ABB RobotStudio station: Lab1.rsstn

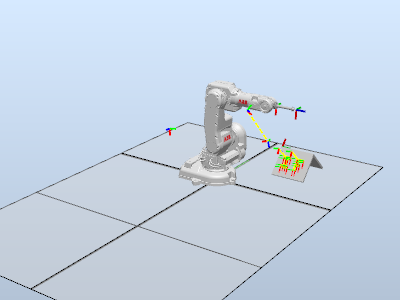
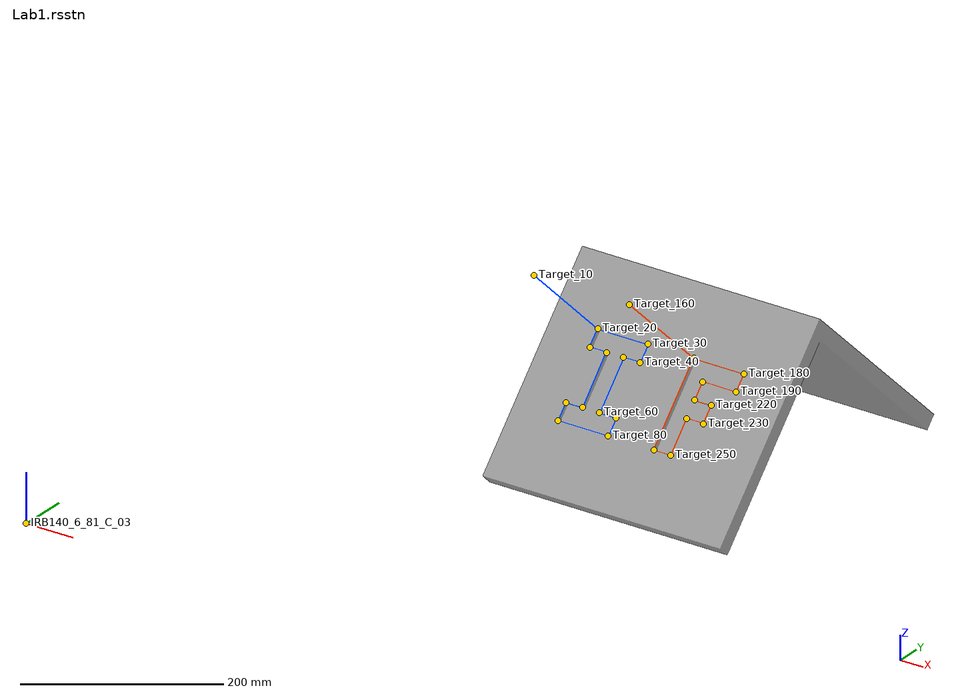
[picture v1: parts stored in the station drawn from their meshes, with robot base, taught points and paths (robot models come from the ABB library and are not in the file)]
Station Station (saved by RobotStudio 22.2.9947.0)
Controller Controlador1
  mechanical unit ROB_1: IRB140_6_81_C_03, 6 joints, base frame (0, 0, 0) mm
Layout (positions relative to the parent item):
  - IRB140_6_81_C_03 [mechanism, from Robots\IRB140_6_81_C_G_03.rslib] at (0, 0, 0) mm; joint values [0, 0, 0, 0, 0, 0] (rad or m)
  - workObjectIF [part] at (600, 500, 191.5) mm, rotated rx -137 ry 0 rz 180 deg, size 284.5 x 267 x 250 mm
  - MarkerIF31 [mechanism] at (515, 0, 712) mm, rotated rx 0 ry 90 rz 0 deg
      TCP MarkerIF31TCP at (-4.09, 34.34, 33.7) mm, rotated rx 0 ry 0 rz -45 deg
      links: tool
Attachment: MarkerIF31 is attached to IRB140_6_81_C_03 / Link6
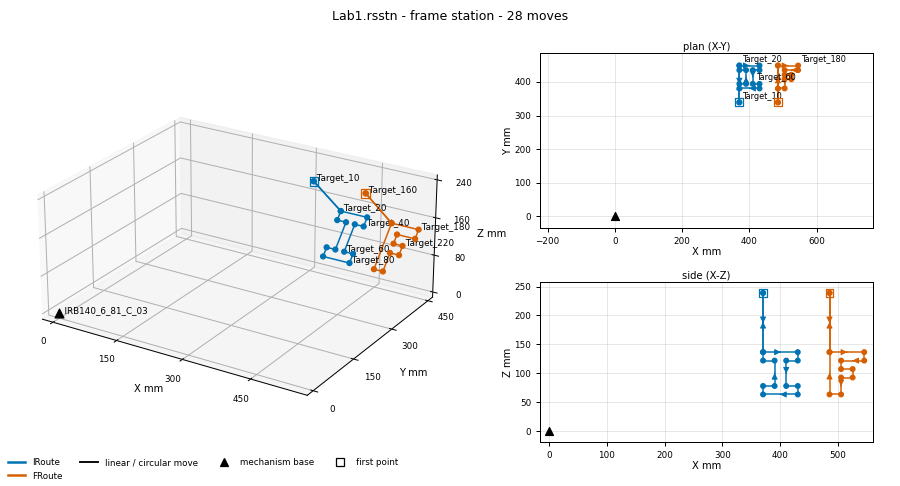
[picture p0: tool path of Lab1.rsstn in frame station, 28 of 32 moves have a stored position in this frame; points joined in program order, loops and branches not executed]
Targets, tools, work objects and paths stored in the station, written as RAPID:
! task T_ROB1
MODULE CalibData
  PERS tooldata MarkerIF31TCP:=[TRUE,[[0,0,164.8],[1,0,0,0]],[1,[0,0,1],[1,0,0,0],0,0,0]];
  TASK PERS wobjdata WOTableIF31:=[FALSE,TRUE,"",[[315.5,500,191.5],[0.281957405,-0.64845973,-0.64845973,-0.281957405]],[[0,0,0],[1,0,0,0]]];
ENDMODULE

! task T_ROB1
MODULE Module1
  CONST robtarget Target_10:=[[-75.000354163,54.833333333,-149.999822918],[0.089424047,0.000001176,0.000000106,0.995993644],[0,0,-2,0],[9E+09,9E+09,9E+09,9E+09,9E+09,9E+09]];
  CONST robtarget Target_20:=[[-75,54.833333333,0.000177081],[0.089424047,0.000001176,0.000000106,0.995993644],[0,1,-2,0],[9E+09,9E+09,9E+09,9E+09,9E+09,9E+09]];
  CONST robtarget Target_30:=[[-75,114.833333333,0.000177081],[0.089424047,0.000001176,0.000000106,0.995993644],[0,0,-2,0],[9E+09,9E+09,9E+09,9E+09,9E+09,9E+09]];
  CONST robtarget Target_40:=[[-95,114.833333333,0.000224303],[0.089424047,0.000001176,0.000000106,0.995993644],[0,1,-2,0],[9E+09,9E+09,9E+09,9E+09,9E+09,9E+09]];
  CONST robtarget Target_50:=[[-95,94.833333333,0.000224303],[0.089424047,0.000001176,0.000000106,0.995993644],[0,1,-2,0],[9E+09,9E+09,9E+09,9E+09,9E+09,9E+09]];
  CONST robtarget Target_60:=[[-155,94.833333333,0.000365968],[0.089424047,0.000001176,0.000000106,0.995993644],[0,1,-2,0],[9E+09,9E+09,9E+09,9E+09,9E+09,9E+09]];
  CONST robtarget Target_70:=[[-155,114.833333333,0.000365968],[0.089424047,0.000001176,0.000000106,0.995993644],[0,1,-2,0],[9E+09,9E+09,9E+09,9E+09,9E+09,9E+09]];
  CONST robtarget Target_80:=[[-174.999999999,114.833333333,0.00041319],[0.089424047,0.000001176,0.000000106,0.995993644],[0,1,-2,0],[9E+09,9E+09,9E+09,9E+09,9E+09,9E+09]];
  CONST robtarget Target_90:=[[-174.999999999,54.833333333,0.00041319],[0.089424047,0.000001176,0.000000106,0.995993644],[0,1,-2,0],[9E+09,9E+09,9E+09,9E+09,9E+09,9E+09]];
  CONST robtarget Target_100:=[[-155,54.833333333,0.000365968],[0.089424047,0.000001176,0.000000106,0.995993644],[0,1,-2,0],[9E+09,9E+09,9E+09,9E+09,9E+09,9E+09]];
  CONST robtarget Target_110:=[[-155,74.833333333,0.000365968],[0.089424047,0.000001176,0.000000106,0.995993644],[0,1,-2,0],[9E+09,9E+09,9E+09,9E+09,9E+09,9E+09]];
  CONST robtarget Target_120:=[[-95,74.833333333,0.000224303],[0.089424047,0.000001176,0.000000106,0.995993644],[0,1,-2,0],[9E+09,9E+09,9E+09,9E+09,9E+09,9E+09]];
  CONST robtarget Target_130:=[[-95,54.833333333,0.000224303],[0.089424047,0.000001176,0.000000106,0.995993644],[0,1,-2,0],[9E+09,9E+09,9E+09,9E+09,9E+09,9E+09]];
  CONST robtarget Target_140:=[[-75,54.833333333,0.000177081],[0.089424047,0.000001176,0.000000106,0.995993644],[0,1,-2,0],[9E+09,9E+09,9E+09,9E+09,9E+09,9E+09]];
  CONST robtarget Target_150:=[[-75.000354163,54.833333333,-149.999822918],[0.089424047,0.000001176,0.000000106,0.995993644],[0,0,-2,0],[9E+09,9E+09,9E+09,9E+09,9E+09,9E+09]];
  CONST robtarget Target_160:=[[-75.000354163,169.666666667,-149.999822918],[0.089424047,0.000001176,0.000000106,0.995993644],[0,0,-2,0],[9E+09,9E+09,9E+09,9E+09,9E+09,9E+09]];
  CONST robtarget Target_170:=[[-75,169.666666667,0.000177081],[0.089424047,0.000001176,0.000000106,0.995993644],[0,0,-2,0],[9E+09,9E+09,9E+09,9E+09,9E+09,9E+09]];
  CONST robtarget Target_180:=[[-75,229.666666667,0.000177081],[0.089424047,0.000001176,0.000000106,0.995993644],[0,0,-2,0],[9E+09,9E+09,9E+09,9E+09,9E+09,9E+09]];
  CONST robtarget Target_190:=[[-95,229.666666667,0.000224303],[0.089424047,0.000001176,0.000000106,0.995993644],[0,0,-2,0],[9E+09,9E+09,9E+09,9E+09,9E+09,9E+09]];
  CONST robtarget Target_200:=[[-95,189.666666667,0.000224303],[0.089424047,0.000001176,0.000000106,0.995993644],[0,0,-2,0],[9E+09,9E+09,9E+09,9E+09,9E+09,9E+09]];
  CONST robtarget Target_210:=[[-114.999999999,189.666666667,0.000271525],[0.089424047,0.000001176,0.000000106,0.995993644],[0,0,-2,0],[9E+09,9E+09,9E+09,9E+09,9E+09,9E+09]];
  CONST robtarget Target_220:=[[-114.999999999,209.666666667,0.000271525],[0.089424047,0.000001176,0.000000106,0.995993644],[0,0,-2,0],[9E+09,9E+09,9E+09,9E+09,9E+09,9E+09]];
  CONST robtarget Target_230:=[[-135,209.666666667,0.000318747],[0.089424047,0.000001176,0.000000106,0.995993644],[0,0,-2,0],[9E+09,9E+09,9E+09,9E+09,9E+09,9E+09]];
  CONST robtarget Target_240:=[[-135,189.666666667,0.000318747],[0.089424047,0.000001176,0.000000106,0.995993644],[0,0,-2,0],[9E+09,9E+09,9E+09,9E+09,9E+09,9E+09]];
  CONST robtarget Target_250:=[[-174.999999999,189.666666667,0.00041319],[0.089424047,0.000001176,0.000000106,0.995993644],[0,0,-2,0],[9E+09,9E+09,9E+09,9E+09,9E+09,9E+09]];
  CONST robtarget Target_260:=[[-174.999999999,169.666666667,0.00041319],[0.089424047,0.000001176,0.000000106,0.995993644],[0,0,-2,0],[9E+09,9E+09,9E+09,9E+09,9E+09,9E+09]];
  CONST robtarget Target_270:=[[-75,169.666666667,0.000177081],[0.089424047,0.000001176,0.000000106,0.995993644],[0,0,-2,0],[9E+09,9E+09,9E+09,9E+09,9E+09,9E+09]];
  CONST robtarget Target_280:=[[-75.000354163,169.666666667,-149.999822918],[0.089424047,0.000001176,0.000000106,0.995993644],[0,0,-2,0],[9E+09,9E+09,9E+09,9E+09,9E+09,9E+09]];
  CONST jointtarget Home:=[[0,0,0,0,0,0],[9E+09,9E+09,9E+09,9E+09,9E+09,9E+09]];
  CONST jointtarget MidPoint:=[[5.481288042,8.647892668,30.215426865,-0.517813809,36.807452266,0],[9E+09,9E+09,9E+09,9E+09,9E+09,9E+09]];
  CONST jointtarget ToolIn:=[[-82.497610687,40.241406603,-45.459191802,6.400380592,0,0],[9E+09,9E+09,9E+09,9E+09,9E+09,9E+09]];
  CONST jointtarget MidMidPoint:=[[-35.566202725,10.598186567,-17.387856543,45.834986846,0,0],[9E+09,9E+09,9E+09,9E+09,9E+09,9E+09]];
  PROC IRoute()
    WaitDI DI_02,1;
    SetDO DO_01,1;
    MoveL Target_10,v150,z10,MarkerIF31TCP\WObj:=WOTableIF31;
    MoveL Target_20,v150,z10,MarkerIF31TCP\WObj:=WOTableIF31;
    MoveL Target_30,v150,z10,MarkerIF31TCP\WObj:=WOTableIF31;
    MoveL Target_40,v150,z10,MarkerIF31TCP\WObj:=WOTableIF31;
    MoveL Target_50,v150,z10,MarkerIF31TCP\WObj:=WOTableIF31;
    MoveL Target_60,v150,z10,MarkerIF31TCP\WObj:=WOTableIF31;
    MoveL Target_70,v150,z10,MarkerIF31TCP\WObj:=WOTableIF31;
    MoveL Target_80,v150,z10,MarkerIF31TCP\WObj:=WOTableIF31;
    MoveL Target_90,v150,z10,MarkerIF31TCP\WObj:=WOTableIF31;
    MoveL Target_100,v150,z10,MarkerIF31TCP\WObj:=WOTableIF31;
    MoveL Target_110,v150,z10,MarkerIF31TCP\WObj:=WOTableIF31;
    MoveL Target_120,v150,z10,MarkerIF31TCP\WObj:=WOTableIF31;
    MoveL Target_130,v150,z10,MarkerIF31TCP\WObj:=WOTableIF31;
    MoveL Target_140,v150,z10,MarkerIF31TCP\WObj:=WOTableIF31;
    MoveL Target_150,v150,z10,MarkerIF31TCP\WObj:=WOTableIF31;
  ENDPROC
  PROC FRoute()
    MoveL Target_160,v150,z5,MarkerIF31TCP\WObj:=WOTableIF31;
    MoveL Target_170,v150,z5,MarkerIF31TCP\WObj:=WOTableIF31;
    MoveL Target_180,v150,z5,MarkerIF31TCP\WObj:=WOTableIF31;
    MoveL Target_190,v150,z5,MarkerIF31TCP\WObj:=WOTableIF31;
    MoveL Target_200,v150,z5,MarkerIF31TCP\WObj:=WOTableIF31;
    MoveL Target_210,v150,z5,MarkerIF31TCP\WObj:=WOTableIF31;
    MoveL Target_220,v150,z5,MarkerIF31TCP\WObj:=WOTableIF31;
    MoveL Target_230,v150,z5,MarkerIF31TCP\WObj:=WOTableIF31;
    MoveL Target_240,v150,z5,MarkerIF31TCP\WObj:=WOTableIF31;
    MoveL Target_250,v150,z5,MarkerIF31TCP\WObj:=WOTableIF31;
    MoveL Target_260,v150,z5,MarkerIF31TCP\WObj:=WOTableIF31;
    MoveL Target_270,v150,z5,MarkerIF31TCP\WObj:=WOTableIF31;
    MoveL Target_280,v150,z5,MarkerIF31TCP\WObj:=WOTableIF31;
    SetDO DO_01,0;
  ENDPROC
  PROC Homing()
    MoveAbsJ Home,v200,z5,MarkerIF31TCP\WObj:=WOTableIF31;
  ENDPROC
  PROC MidGoing()
    WaitDI DI_01,1;
    MoveAbsJ MidMidPoint,v200,z5,MarkerIF31TCP\WObj:=WOTableIF31;
    MoveAbsJ MidPoint,v200,z5,MarkerIF31TCP\WObj:=WOTableIF31;
  ENDPROC
  PROC ToolMoving()
    MoveAbsJ ToolIn,v200,z5,MarkerIF31TCP\WObj:=WOTableIF31;
  ENDPROC
ENDMODULE

